Staubli VAL3: extAxisCan.dtx

public aio aiPosFbk = {link=CanIO\Axis7\drvPosFbk_0}
public aio aoIPPos = {link=CanIO\Axis7\drvIPCmdPos_0}
public aio aoIPSpd = {link=CanIO\Axis7\ipVel_0}
public aio aoPosCmd = {link=CanIO\Axis7\drvCmdPos_0}
public aio aoWorkMode = {link=CanIO\Axis7\drvworkmode}
public bool bDriveQuickStop
public bool bDrivesOpEnable
bool bDrivesSwOnDis
public bool bDrvFault[2]
bool bEnableRequest
bool bIsS7_6 = true
bool bMemPower
public bool bNoDrivesFault = true
public bool bOpeEnabled[2]
bool bOverrun
public bool bQuickStop[2]
public bool bSWOnDis
public bool bSysShut
public bool blifebit[2]
  [0] = true
  [1] = true
bool blifebit_all_ok = true
public dio diFault = {link=CanIO\Axis7\fault_0}
public dio diHomingError = {link=CanIO\Axis7\homingError_0}
public dio diHomingReached = {link=CanIO\Axis7\homingReached_0}
public dio diIntLmtAct = {link=CanIO\Axis7\intLmtAct_0}
public dio diOpeEnabled = {link=CanIO\Axis7\opeEnabled_0}
public dio diPosReached = {link=CanIO\Axis7\targetReached_0}
public dio diQuickStop = {link=CanIO\Axis7\quickStopped_0}
public dio diReady2SwOn = {link=CanIO\Axis7\ready2SwOn_0}
public dio diSwOnDis = {link=CanIO\Axis7\swOnDis_0}
public dio diSwitchedOn = {link=CanIO\Axis7\switchedOn_0}
public dio diTargetReach = {link=CanIO\Axis7\targetReached_0}
public dio diVoltEnabled = {link=CanIO\Axis7\voltEnabled_0}
public dio diWarning = {link=CanIO\Axis7\warning_0}
public dio doEnableOp = {link=CanIO\Axis7\enableOp_0}
public dio doEnableVoltage = {link=CanIO\Axis7\enableVolt_0}
public dio doFaultReset = {link=CanIO\Axis7\faultReset_0}
public dio doManual = {link=CanIO\Axis7\Manual}
public dio doQuickStop = {link=CanIO\Axis7\quickStop_0}
public dio doStartHoming = {link=CanIO\Axis7\startHoming_0}
public dio doSwitchOn = {link=CanIO\Axis7\switchOn_0}
jointRx jDummy = {j1=1.48, j2=0.75, j3=2.04, j4=1.56, j5=2.81, j6=1.79}
jointRx jPosErrMax = {j1=100, j2=100, j3=100, j4=100, j5=100, j6=100}
jointRx jZero = {j1=0.01, j2=0.01, j3=0.01, j4=0.01, j5=0.01, j6=0.01}
public num nAxesPosFbk[2]
public num nAxesSum = 2
num nCntDrvDisable
num nCntDrvEnable[2]
public num nDrvFbkPos[2]
num nDrvPos[2]
num nDrvState[2]
  [0] = 1
  [1] = 1
public num nExtAxseAccDft = 10
public num nExtAxseSpdDft = 10
num nGearratio[2]
  [0] = 10
  [1] = 1
public num nResolution[2]
  [0] = 1280000
  [1] = 180000
public num nScaleFact[2]
  [0] = 10
  [1] = 360
public string sMsg
string sVersion = "s7.6 - May 29 2013 - 16:53:12"
public dio diRemote = {link=CanIO\Axis7\remote_0}
num nManul = 10
num nBuffSize
num nAxesData
public bool bMoveType
frame fFrame = {fatherId=world[0]}
